// TIA Portal V17 export
// export: Created 2022-07-28T18:02:47.4319373Z, ExportSetting None, DisplayName Totally Integrated Automation Portal, DisplayVersion V17, DisplayName TIA Portal Openness, DisplayVersion V17, DisplayName TIA Portal Teamcenter Gateway, DisplayVersion V17, DisplayName TIA Portal Version Control Interface, DisplayVersion V17, DisplayName TIA Portal Test Suite Advanced, DisplayVersion V17, DisplayName SINAMICS Startdrive Advanced, DisplayVersion V17, DisplayName SINAMICS DCC, DisplayVersion V17, DisplayName SINAMICS Startdrive G130, G150, S120, S150, SINAMICS MV, S210, DisplayVersion V17, DisplayName SINAMICS Startdrive G110M, G120, G120C, G120D, G120P, G115D, DisplayVersion V17, DisplayName STEP 7 Professional, DisplayVersion V17, DisplayName SIMATIC Energy Suite, DisplayVersion V17, DisplayName STEP 7 CFC, DisplayVersion V17, DisplayName STEP 7 Safety, DisplayVersion V17, DisplayName WinCC Advanced / Unified PC, DisplayVersion V17, DisplayName SIMATIC Visualization Architect, DisplayVersion V17
FUNCTION "H02_FC" : Void   // FC15, SCL
{ S7_Optimized_Access := 'TRUE' }
// stored: SetENOAutomatically false
   VAR_TEMP
      t_SupplyRelease : Bool;   // 1 - Release from supply
   END_VAR
BEGIN
   #t_SupplyRelease := true;

   REGION (ID = 14) Насос оборотної води 1 Н1Гр
       //Тип елемента: Насос з ПЧ
       //Параметри двигуна: P=75kW;V=400V;I=133A;f=0.86;v=2979rpm;
       //Параметри ПЧ: G120C; Profinet = 8 Words;

       REGION Блокування та зовнішні аварії
           REGION Блокування forward
               "D_N1Gr_Ctrl".IB_InterlocksForward_8.%X0 := false;
               "D_N1Gr_Ctrl".IB_InterlocksForward_8.%X1 := false;
               "D_N1Gr_Ctrl".IB_InterlocksForward_8.%X2 := false;
               "D_N1Gr_Ctrl".IB_InterlocksForward_8.%X3 := false;
               "D_N1Gr_Ctrl".IB_InterlocksForward_8.%X4 := false;
               "D_N1Gr_Ctrl".IB_InterlocksForward_8.%X5 := false;
               "D_N1Gr_Ctrl".IB_InterlocksForward_8.%X6 := false;
               "D_N1Gr_Ctrl".IB_InterlocksForward_8.%X7 := false;
           END_REGION

           REGION Блокування reverse
               "D_N1Gr_Ctrl".IB_InterlocksReverse_8.%X0 := false;
               "D_N1Gr_Ctrl".IB_InterlocksReverse_8.%X1 := false;
               "D_N1Gr_Ctrl".IB_InterlocksReverse_8.%X2 := false;
               "D_N1Gr_Ctrl".IB_InterlocksReverse_8.%X3 := false;
               "D_N1Gr_Ctrl".IB_InterlocksReverse_8.%X4 := false;
               "D_N1Gr_Ctrl".IB_InterlocksReverse_8.%X5 := false;
               "D_N1Gr_Ctrl".IB_InterlocksReverse_8.%X6 := false;
               "D_N1Gr_Ctrl".IB_InterlocksReverse_8.%X7 := false;
           END_REGION

           REGION Зовнішні аварії та попередження
               "D_N1Gr_Ctrl".IW_ExternalError_16.%X0 := false;
               "D_N1Gr_Ctrl".IW_ExternalError_16.%X1 := false;
               "D_N1Gr_Ctrl".IW_ExternalError_16.%X2 := false;
               "D_N1Gr_Ctrl".IW_ExternalError_16.%X3 := false;
               "D_N1Gr_Ctrl".IW_ExternalError_16.%X4 := false;
               "D_N1Gr_Ctrl".IW_ExternalError_16.%X5 := false;
               "D_N1Gr_Ctrl".IW_ExternalError_16.%X6 := false;
               "D_N1Gr_Ctrl".IW_ExternalError_16.%X7 := false;
               "D_N1Gr_Ctrl".IW_ExternalError_16.%X8 := false;
               "D_N1Gr_Ctrl".IW_ExternalError_16.%X9 := false;
               "D_N1Gr_Ctrl".IW_ExternalError_16.%X10 := false;
               "D_N1Gr_Ctrl".IW_ExternalError_16.%X11 := false;
               "D_N1Gr_Ctrl".IW_ExternalError_16.%X12 := false;
               "D_N1Gr_Ctrl".IW_ExternalError_16.%X13 := false;
               "D_N1Gr_Ctrl".IW_ExternalError_16.%X14 := false;
               "D_N1Gr_Ctrl".IW_ExternalError_16.%X15 := false;

               "D_N1Gr_Ctrl".I_ExternalWarning := false;
           END_REGION
       END_REGION

       REGION Блок керування
           "D_N1Gr_Ctrl"(I_Initialization := "D_General_ProgramDATA".RestartPLC,
                         IR_CycleTime := "D_PLC".TIME_TCK.cyclic_sec_R,
                         II_Obj_ID := 14,
                         I_CmdGeneralReset := "D_General_ProgramDATA".ResetGlobal,
                         I_One_1s := "D_PLC".PLS.P1S,
                         I_EnableHorn := false,
                         I_EstopLocal := "D_InOut"."N1Gr".I_ES,
                         I_EstopHMI := "D_General_ProgramDATA".ES_HMI_Global
                         AND "D_General_ProgramDATA".ES_Fld_Global,
                         I_SuppyBox_Ok := #t_SupplyRelease,
                         I_MP_Ok := "D_InOut"."N1Gr".I_MCP,
                         I_ThermoDefend := true,
                         I_TripBus:="D_PN_IO_Status".States_Proc[1],
                         I_Termistor_Ok := "D_InOut"."N1Gr".I_PTC_Ok,
                         IR_TimeTripInverter:=30.0,
                         IQ_PLC_CycleInfo := "D_PLC_CycleInfo_DATA".Grp_Obj[1, 0]);
       END_REGION

       REGION Блок частотного перетворювача
           "D_N1Gr_Inv"(II_Obj_ID := 14,
                        I_HW_Tel_ID := 301);
       END_REGION

   END_REGION
END_FUNCTION
